(* PLC project 117_1_V0.5.project, CODESYS CODESYS V3.5 SP17 Patch 3 *)
(* stored: creationDateTime 1970-01-01T00:00:00, modificationDateTime 2026-06-16T22:51:19.9979415 *)

FUNCTION_BLOCK TestingForces_53868
  VAR_INPUT
    P : E_P1_2;
    I_II : E_I_II;
  END_VAR
  VAR_OUTPUT
    Fstab : UDINT;
    Fset : UDINT;
    Fsp : UDINT;
    F_su_lower_level : UDINT;
    F_su_upper_level : UDINT;
  END_VAR

            CASE P OF
	
	P1:
		CASE I_II OF
			I: 
				Fstab				:= 50;
// 				Fset				:= 736;
// 				Fsp					:= 1610;	
 				F_su_lower_level	:= 930;		
				F_su_upper_level	:= 1240;
			II:   
				Fstab				:= 50;
// 				Fset				:= 638; 
// 				Fsp					:= 1395;
				F_su_lower_level	:= 825;
				F_su_upper_level	:= 1100;
		END_CASE
		
	P2:
		CASE I_II OF
			I: 
				Fstab				:= 50;
// 				Fset				:= 944; 
// 				Fsp					:= 2065;
				F_su_lower_level	:= 1680;
				F_su_upper_level	:= 2250;
			II: 
				Fstab				:= 50;
// 				Fset				:= 828; 
// 				Fsp					:= 1811; 
				F_su_lower_level	:= 1490;
				F_su_upper_level	:= 1990;
		END_CASE
END_CASE
          
END_FUNCTION_BLOCK
